PROGRAM VGR_State
VAR
	
	bStateIdle: BOOL := TRUE;
	bStatePlace: BOOL;
	bStateHoming: BOOL;
	bStatePick: BOOL;
	tolerance : UINT := 5;
	
	bInPositionPickVertical : BOOL;
	bInPositionPickHorizontal : BOOL;
	bInPositionPickRotate : BOOL;
	bInPositionPlaceVertical : BOOL;
	bInPositionPlaceHorizontal : BOOL;
	bInPositionPlaceRotate : BOOL;
	
	bValveClosed : BOOL;
	
	RS_Idle: RS;
	
	RS_Homing: RS;
	
	RS_Pick: RS;
	bValveOpened: BOOL;
	RS_Place: RS;
	bValveOpen: BOOL;
	SR_ESTOP: SR;
	bStateEStop: BOOL;
	AxisMovementController_Vertical: AxisMovementController;
	AxisMovementController_Horizontal: AxisMovementController;
	AxisReferencing_Vertical: AxisReferencing;
	AxisReferencing_Horizontal: AxisReferencing;
	AxisReferencing_Rotational: AxisReferencing;
	AxisMovementController_Rotation: AxisMovementController;
END_VAR
VAR // added by the converter: edge detectors and wires of the graphical bodies
    _w1 : BOOL;
END_VAR

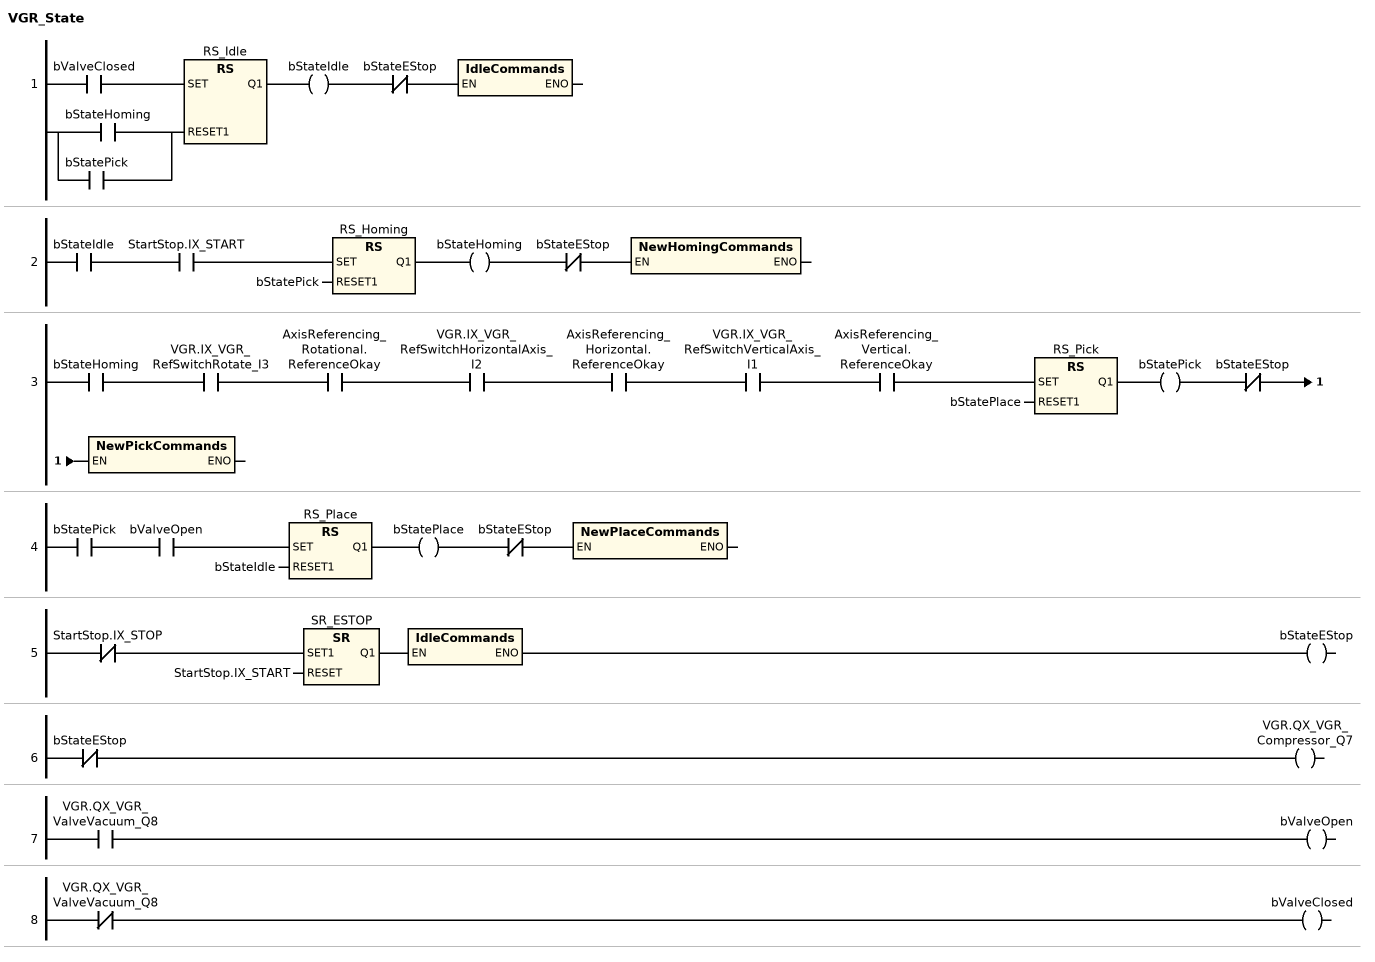
// NETWORK 1
RS_Idle(SET := bValveClosed, RESET1 := bStateHoming OR bStatePick); // RS
bStateIdle := RS_Idle.Q1;
IF RS_Idle.Q1 AND NOT bStateEStop THEN IdleCommands(); END_IF

// NETWORK 2
RS_Homing(SET := bStateIdle AND StartStop.IX_START, RESET1 := bStatePick); // RS
bStateHoming := RS_Homing.Q1;
IF RS_Homing.Q1 AND NOT bStateEStop THEN NewHomingCommands(); END_IF

// NETWORK 3
RS_Pick(SET := bStateHoming AND VGR.IX_VGR_RefSwitchRotate_I3 AND AxisReferencing_Rotational.ReferenceOkay AND VGR.IX_VGR_RefSwitchHorizontalAxis_I2 AND AxisReferencing_Horizontal.ReferenceOkay AND VGR.IX_VGR_RefSwitchVerticalAxis_I1 AND AxisReferencing_Vertical.ReferenceOkay, RESET1 := bStatePlace); // RS
bStatePick := RS_Pick.Q1;
IF RS_Pick.Q1 AND NOT bStateEStop THEN NewPickCommands(); END_IF

// NETWORK 4
RS_Place(SET := bStatePick AND bValveOpen, RESET1 := bStateIdle); // RS
bStatePlace := RS_Place.Q1;
IF RS_Place.Q1 AND NOT bStateEStop THEN NewPlaceCommands(); END_IF

// NETWORK 5
SR_ESTOP(SET1 := NOT StartStop.IX_STOP, RESET := StartStop.IX_START); // SR
_w1 := SR_ESTOP.Q1;
IF _w1 THEN IdleCommands(); END_IF
bStateEStop := _w1;

// NETWORK 6
VGR.QX_VGR_Compressor_Q7 := NOT bStateEStop;

// NETWORK 7
bValveOpen := VGR.QX_VGR_ValveVacuum_Q8;

// NETWORK 8
bValveClosed := NOT VGR.QX_VGR_ValveVacuum_Q8;

ACTION HomeCommands:
IF VGR.IX_VGR_RefSwitchVerticalAxis_I1 THEN
	VGR.QX_VGR_M1_VerticalAxisUp_Q1 := FALSE;
	VGR.QX_VGR_M1_VerticalAxisDown_Q2 := FALSE;
	VGR.QW_VGR_PWM_Vertical_Control := 0;
	VGR.QW_VGR_PWM_Vertical_M1 := 0;
	Encoder.setCounterVertical := TRUE;
	Encoder.setCounterValueVertical:= 0;
ELSE
	VGR.QX_VGR_M1_VerticalAxisUp_Q1 := TRUE;
	VGR.QX_VGR_M1_VerticalAxisDown_Q2 := FALSE;
	VGR.QW_VGR_PWM_Vertical_Control := 32;
	VGR.QW_VGR_PWM_Vertical_M1 := 5000;
END_IF
IF VGR.IX_VGR_RefSwitchHorizontalAxis_I2 THEN
	VGR.QX_VGR_M2_HorizontalAxisBackward_Q3 := FALSE;
    VGR.QX_VGR_M2_HorizontalAxisForward_Q4 := FALSE;
    VGR.QW_VGR_PWM_Horizontal_Control := 0;
    VGR.QW_VGR_PWM_Horizontal_M2 := 0;
	Encoder.setCounterHorizontal := TRUE;
ELSE
	VGR.QX_VGR_M2_HorizontalAxisBackward_Q3 := TRUE;
    VGR.QX_VGR_M2_HorizontalAxisForward_Q4 := FALSE;
    VGR.QW_VGR_PWM_Horizontal_Control := 32;
    VGR.QW_VGR_PWM_Horizontal_M2 := 5000;
END_IF
IF VGR.IX_VGR_RefSwitchHorizontalAxis_I2 THEN
	VGR.QX_VGR_M3_RotateClockwise_Q5 := FALSE;
    VGR.QX_VGR_M3_RotateCounterClockwise_Q6 := FALSE;
    VGR.QW_VGR_PWM_Rotate_Control := 0;
    VGR.QW_VGR_PWM_Rotate_M3 := 0;
	Encoder.setCounterRotate := TRUE;
ELSE
	VGR.QX_VGR_M3_RotateClockwise_Q5 := TRUE;
    VGR.QX_VGR_M3_RotateCounterClockwise_Q6 := FALSE;
    VGR.QW_VGR_PWM_Rotate_Control := 32;
    VGR.QW_VGR_PWM_Rotate_M3 := 5000;
END_IF
END_ACTION

ACTION IdleCommands:
VGR.QX_VGR_M1_VerticalAxisUp_Q1 := FALSE;
VGR.QX_VGR_M1_VerticalAxisDown_Q2 := FALSE;
VGR.QW_VGR_PWM_Vertical_Control := 0;
VGR.QW_VGR_PWM_Vertical_M1 := 0;
VGR.QX_VGR_M2_HorizontalAxisBackward_Q3 := FALSE;
VGR.QX_VGR_M2_HorizontalAxisForward_Q4 := FALSE;
VGR.QW_VGR_PWM_Horizontal_Control := 0;
VGR.QW_VGR_PWM_Horizontal_M2 := 0;
VGR.QX_VGR_M3_RotateClockwise_Q5 := FALSE;
VGR.QX_VGR_M3_RotateCounterClockwise_Q6 := FALSE;
VGR.QW_VGR_PWM_Rotate_Control := 0;
VGR.QW_VGR_PWM_Rotate_M3 := 0;
END_ACTION

ACTION NewHomingCommands:
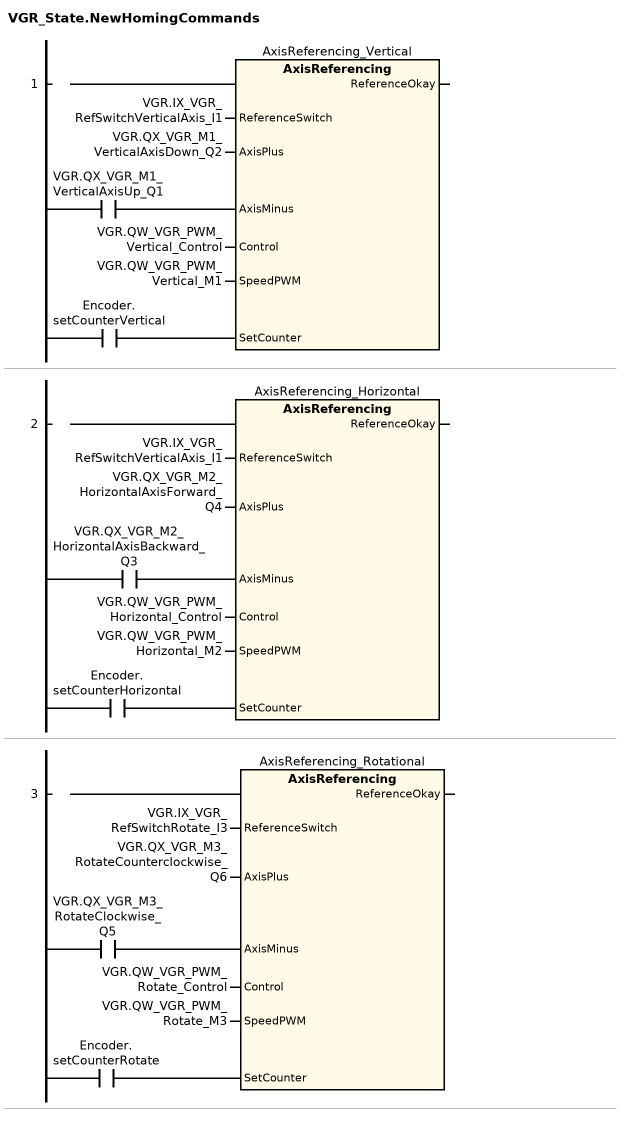
// NETWORK 1
AxisReferencing_Vertical(
    ReferenceSwitch := VGR.IX_VGR_RefSwitchVerticalAxis_I1,
    AxisPlus := VGR.QX_VGR_M1_VerticalAxisDown_Q2,
    AxisMinus := VGR.QX_VGR_M1_VerticalAxisUp_Q1,
    Control := VGR.QW_VGR_PWM_Vertical_Control,
    SpeedPWM := VGR.QW_VGR_PWM_Vertical_M1,
    SetCounter := Encoder.setCounterVertical); // AxisReferencing

// NETWORK 2
AxisReferencing_Horizontal(
    ReferenceSwitch := VGR.IX_VGR_RefSwitchVerticalAxis_I1,
    AxisPlus := VGR.QX_VGR_M2_HorizontalAxisForward_Q4,
    AxisMinus := VGR.QX_VGR_M2_HorizontalAxisBackward_Q3,
    Control := VGR.QW_VGR_PWM_Horizontal_Control,
    SpeedPWM := VGR.QW_VGR_PWM_Horizontal_M2,
    SetCounter := Encoder.setCounterHorizontal); // AxisReferencing

// NETWORK 3
AxisReferencing_Rotational(
    ReferenceSwitch := VGR.IX_VGR_RefSwitchRotate_I3,
    AxisPlus := VGR.QX_VGR_M3_RotateCounterclockwise_Q6,
    AxisMinus := VGR.QX_VGR_M3_RotateClockwise_Q5,
    Control := VGR.QW_VGR_PWM_Rotate_Control,
    SpeedPWM := VGR.QW_VGR_PWM_Rotate_M3,
    SetCounter := Encoder.setCounterRotate); // AxisReferencing
END_ACTION

ACTION NewPickCommands:
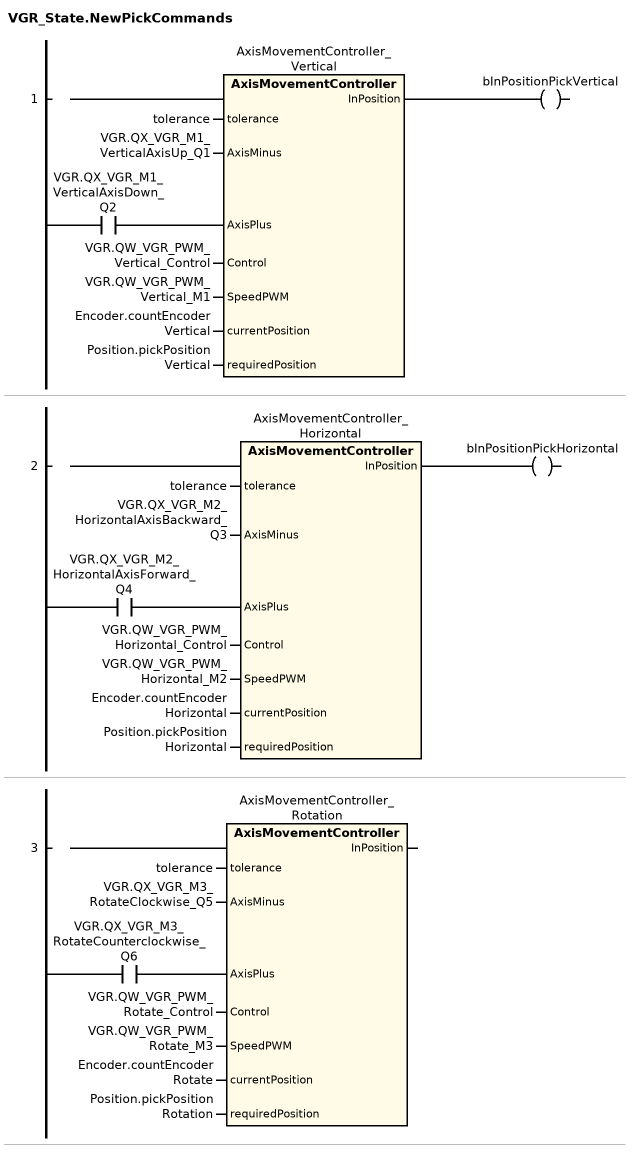
// NETWORK 1
AxisMovementController_Vertical(
    tolerance := tolerance,
    AxisMinus := VGR.QX_VGR_M1_VerticalAxisUp_Q1,
    AxisPlus := VGR.QX_VGR_M1_VerticalAxisDown_Q2,
    Control := VGR.QW_VGR_PWM_Vertical_Control,
    SpeedPWM := VGR.QW_VGR_PWM_Vertical_M1,
    currentPosition := Encoder.countEncoderVertical,
    requiredPosition := Position.pickPositionVertical); // AxisMovementController
bInPositionPickVertical := AxisMovementController_Vertical.InPosition;

// NETWORK 2
AxisMovementController_Horizontal(
    tolerance := tolerance,
    AxisMinus := VGR.QX_VGR_M2_HorizontalAxisBackward_Q3,
    AxisPlus := VGR.QX_VGR_M2_HorizontalAxisForward_Q4,
    Control := VGR.QW_VGR_PWM_Horizontal_Control,
    SpeedPWM := VGR.QW_VGR_PWM_Horizontal_M2,
    currentPosition := Encoder.countEncoderHorizontal,
    requiredPosition := Position.pickPositionHorizontal); // AxisMovementController
bInPositionPickHorizontal := AxisMovementController_Horizontal.InPosition;

// NETWORK 3
AxisMovementController_Rotation(
    tolerance := tolerance,
    AxisMinus := VGR.QX_VGR_M3_RotateClockwise_Q5,
    AxisPlus := VGR.QX_VGR_M3_RotateCounterclockwise_Q6,
    Control := VGR.QW_VGR_PWM_Rotate_Control,
    SpeedPWM := VGR.QW_VGR_PWM_Rotate_M3,
    currentPosition := Encoder.countEncoderRotate,
    requiredPosition := Position.pickPositionRotation); // AxisMovementController
END_ACTION

ACTION NewPlaceCommands:
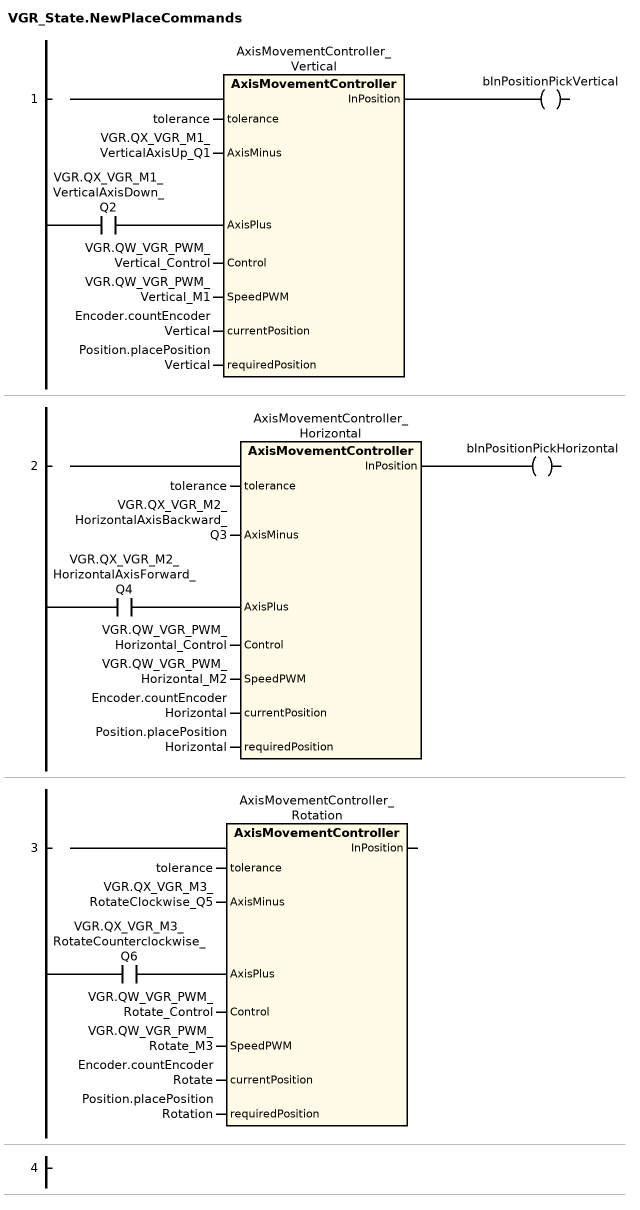
// NETWORK 1
AxisMovementController_Vertical(
    tolerance := tolerance,
    AxisMinus := VGR.QX_VGR_M1_VerticalAxisUp_Q1,
    AxisPlus := VGR.QX_VGR_M1_VerticalAxisDown_Q2,
    Control := VGR.QW_VGR_PWM_Vertical_Control,
    SpeedPWM := VGR.QW_VGR_PWM_Vertical_M1,
    currentPosition := Encoder.countEncoderVertical,
    requiredPosition := Position.placePositionVertical); // AxisMovementController
bInPositionPickVertical := AxisMovementController_Vertical.InPosition;

// NETWORK 2
AxisMovementController_Horizontal(
    tolerance := tolerance,
    AxisMinus := VGR.QX_VGR_M2_HorizontalAxisBackward_Q3,
    AxisPlus := VGR.QX_VGR_M2_HorizontalAxisForward_Q4,
    Control := VGR.QW_VGR_PWM_Horizontal_Control,
    SpeedPWM := VGR.QW_VGR_PWM_Horizontal_M2,
    currentPosition := Encoder.countEncoderHorizontal,
    requiredPosition := Position.placePositionHorizontal); // AxisMovementController
bInPositionPickHorizontal := AxisMovementController_Horizontal.InPosition;

// NETWORK 3
AxisMovementController_Rotation(
    tolerance := tolerance,
    AxisMinus := VGR.QX_VGR_M3_RotateClockwise_Q5,
    AxisPlus := VGR.QX_VGR_M3_RotateCounterclockwise_Q6,
    Control := VGR.QW_VGR_PWM_Rotate_Control,
    SpeedPWM := VGR.QW_VGR_PWM_Rotate_M3,
    currentPosition := Encoder.countEncoderRotate,
    requiredPosition := Position.placePositionRotation); // AxisMovementController

// NETWORK 4
END_ACTION

ACTION PickCommands:
IF  AboutEqual(IN1:= Encoder.countEncoderVertical,
	IN2:= Position.pickPositionVertical,
Tolerance:= tolerance)
 THEN
	VGR.QX_VGR_M1_VerticalAxisUp_Q1 := FALSE;
	VGR.QX_VGR_M1_VerticalAxisDown_Q2 := FALSE;
	VGR.QW_VGR_PWM_Vertical_Control := 0;
	VGR.QW_VGR_PWM_Vertical_M1 := 0;
	bInPositionPickVertical := TRUE;
ELSIF Encoder.countEncoderVertical > Position.pickPositionVertical AND NOT bInPositionPickVertical THEN
	VGR.QX_VGR_M1_VerticalAxisUp_Q1 := TRUE;
	VGR.QX_VGR_M1_VerticalAxisDown_Q2 := FALSE;
	VGR.QW_VGR_PWM_Vertical_Control := 32;
	VGR.QW_VGR_PWM_Vertical_M1 := 5000;
	bInPositionPickVertical := FALSE;
ELSE
	VGR.QX_VGR_M1_VerticalAxisUp_Q1 := FALSE;
	VGR.QX_VGR_M1_VerticalAxisDown_Q2 := TRUE;
	VGR.QW_VGR_PWM_Vertical_Control := 32;
	VGR.QW_VGR_PWM_Vertical_M1 := 5000;
	bInPositionPickVertical := FALSE;
END_IF
IF AboutEqual(IN1:= Encoder.countEncoderHorizontal,
	IN2:= Position.pickPositionHorizontal,
Tolerance:= tolerance) THEN
	VGR.QX_VGR_M2_HorizontalAxisBackward_Q3 := FALSE;
    VGR.QX_VGR_M2_HorizontalAxisForward_Q4 := FALSE;
    VGR.QW_VGR_PWM_Horizontal_Control := 0;
    VGR.QW_VGR_PWM_Horizontal_M2 := 0;
	bInPositionPickHorizontal := TRUE;
ELSIF Encoder.countEncoderHorizontal > Position.pickPositionHorizontal  AND NOT bInPositionPickHorizontal THEN
	VGR.QX_VGR_M2_HorizontalAxisBackward_Q3 := TRUE;
    VGR.QX_VGR_M2_HorizontalAxisForward_Q4 := FALSE;
    VGR.QW_VGR_PWM_Horizontal_Control := 32;
    VGR.QW_VGR_PWM_Horizontal_M2 := 5000;
	bInPositionPickHorizontal := FALSE;
ELSE
	VGR.QX_VGR_M2_HorizontalAxisBackward_Q3 := FALSE;
	VGR.QX_VGR_M2_HorizontalAxisForward_Q4 := TRUE;
	VGR.QW_VGR_PWM_Horizontal_Control := 32;
	VGR.QW_VGR_PWM_Horizontal_M2 := 5000;
	bInPositionPickHorizontal := FALSE;
END_IF
IF  AboutEqual(IN1:= Encoder.countEncoderRotate,
	IN2:= Position.pickPositionRotation,
Tolerance:= tolerance) THEN
    VGR.QX_VGR_M3_RotateClockwise_Q5 := FALSE;
    VGR.QX_VGR_M3_RotateCounterClockwise_Q6 := FALSE;
    VGR.QW_VGR_PWM_Rotate_Control := 0;
    VGR.QW_VGR_PWM_Rotate_M3 := 0;
	bInPositionPickRotate := TRUE;
ELSIF Encoder.countEncoderRotate > Position.pickPositionRotation  AND NOT bInPositionPickRotate THEN
	VGR.QX_VGR_M3_RotateClockwise_Q5 := FALSE;
    VGR.QX_VGR_M3_RotateCounterClockwise_Q6 := TRUE;
    VGR.QW_VGR_PWM_Rotate_Control := 32;
    VGR.QW_VGR_PWM_Rotate_M3 := 5000;
	bInPositionPickRotate := FALSE;
ELSE
	VGR.QX_VGR_M3_RotateClockwise_Q5 := TRUE;
    VGR.QX_VGR_M3_RotateCounterClockwise_Q6 := FALSE;
    VGR.QW_VGR_PWM_Rotate_Control := 32;
    VGR.QW_VGR_PWM_Rotate_M3 := 5000;
	bInPositionPickRotate := FALSE;
END_IF

IF bInPositionPickRotate AND bInPositionPickRotate AND bInPositionPickRotate THEN
	VGR.QX_VGR_ValveVacuum_Q8 := TRUE;
ELSE
	VGR.QX_VGR_ValveVacuum_Q8 := FALSE;
END_IF
END_ACTION

ACTION PlaceCommands:
IF  Encoder.countEncoderVertical = Position.placePositionVertical OR
	(Position.pickPositionVertical+tolerance > Encoder.countEncoderVertical OR 
	Encoder.countEncoderVertical > Position.pickPositionVertical-tolerance ) THEN
	VGR.QX_VGR_M1_VerticalAxisUp_Q1 := FALSE;
	VGR.QX_VGR_M1_VerticalAxisDown_Q2 := FALSE;
	VGR.QW_VGR_PWM_Vertical_Control := 0;
	VGR.QW_VGR_PWM_Vertical_M1 := 0;
	bInPositionPlaceVertical := TRUE;
ELSIF Encoder.countEncoderVertical > Position.placePositionVertical THEN
	VGR.QX_VGR_M1_VerticalAxisUp_Q1 := FALSE;
	VGR.QX_VGR_M1_VerticalAxisDown_Q2 := TRUE;
	VGR.QW_VGR_PWM_Vertical_Control := 32;
	VGR.QW_VGR_PWM_Vertical_M1 := 5000;
	bInPositionPlaceVertical := FALSE;
ELSE
	VGR.QX_VGR_M1_VerticalAxisUp_Q1 := TRUE;
	VGR.QX_VGR_M1_VerticalAxisDown_Q2 := FALSE;
	VGR.QW_VGR_PWM_Vertical_Control := 32;
	VGR.QW_VGR_PWM_Vertical_M1 := 5000;
	bInPositionPlaceVertical := FALSE;
END_IF
IF Encoder.countEncoderHorizontal = Position.placePositionHorizontal OR 
(Encoder.countEncoderHorizontal < Position.pickPositionHorizontal + tolerance)OR 
(Encoder.countEncoderHorizontal > Position.pickPositionHorizontal -tolerance) THEN
	VGR.QX_VGR_M2_HorizontalAxisBackward_Q3 := FALSE;
    VGR.QX_VGR_M2_HorizontalAxisForward_Q4 := FALSE;
    VGR.QW_VGR_PWM_Horizontal_Control := 0;
    VGR.QW_VGR_PWM_Horizontal_M2 := 0;
	bInPositionPlaceHorizontal := TRUE;
ELSIF Encoder.countEncoderHorizontal > Position.placePositionHorizontal THEN
	VGR.QX_VGR_M2_HorizontalAxisBackward_Q3 := TRUE;
    VGR.QX_VGR_M2_HorizontalAxisForward_Q4 := FALSE;
    VGR.QW_VGR_PWM_Horizontal_Control := 32;
    VGR.QW_VGR_PWM_Horizontal_M2 := 5000;
	bInPositionPlaceHorizontal := FALSE;
ELSE
	VGR.QX_VGR_M2_HorizontalAxisBackward_Q3 := FALSE;
	VGR.QX_VGR_M2_HorizontalAxisForward_Q4 := TRUE;
	VGR.QW_VGR_PWM_Horizontal_Control := 32;
	VGR.QW_VGR_PWM_Horizontal_M2 := 5000;
	bInPositionPlaceHorizontal := FALSE;
END_IF
IF  Encoder.countEncoderRotate=Position.placePositionRotation  OR 
(Encoder.countEncoderRotate < Position.pickPositionRotation+tolerance) OR 
(Encoder.countEncoderRotate>Position.pickPositionRotation-tolerance) THEN
    VGR.QX_VGR_M3_RotateClockwise_Q5 := FALSE;
    VGR.QX_VGR_M3_RotateCounterClockwise_Q6 := FALSE;
    VGR.QW_VGR_PWM_Rotate_Control := 0;
    VGR.QW_VGR_PWM_Rotate_M3 := 0;
	bInPositionPlaceRotate := TRUE;
ELSIF Encoder.countEncoderRotate > Position.placePositionRotation THEN
	VGR.QX_VGR_M3_RotateClockwise_Q5 := FALSE;
    VGR.QX_VGR_M3_RotateCounterClockwise_Q6 := TRUE;
    VGR.QW_VGR_PWM_Rotate_Control := 32;
    VGR.QW_VGR_PWM_Rotate_M3 := 5000;
	bInPositionPlaceRotate := FALSE;
ELSE
	VGR.QX_VGR_M3_RotateClockwise_Q5 := TRUE;
    VGR.QX_VGR_M3_RotateCounterClockwise_Q6 := FALSE;
    VGR.QW_VGR_PWM_Rotate_Control := 32;
    VGR.QW_VGR_PWM_Rotate_M3 := 5000;
	bInPositionPlaceRotate := FALSE;
END_IF

IF bInPositionPlaceHorizontal AND bInPositionPlaceRotate AND bInPositionPlaceVertical THEN
	VGR.QX_VGR_ValveVacuum_Q8 := FALSE;
ELSE
	VGR.QX_VGR_ValveVacuum_Q8 := TRUE;
END_IF
END_ACTION

END_PROGRAM

(* stored: Version 1.1.0.1, ProductVersion 3.1.4024.12
   POU VGR_State: Id {7aa8a406-b458-426c-9530-cc62a1b42f8a}, SpecialFunc None
   Action HomeCommands: Id {0f636ef8-07f3-4884-a7a6-370109e8cfaa}
   Action IdleCommands: Id {c22b6015-031e-44d1-9a49-ef0c9e3c7f44}
   Action NewHomingCommands: Id {56950258-6488-4c40-9d15-434b1ca9d02a}
   Action NewPickCommands: Id {c336029e-b54d-4c80-b2f9-8cac11d6896b}
   Action NewPlaceCommands: Id {43b75217-0a31-4d31-9610-cf6accadfee8}
   Action PickCommands: Id {dc673986-ad1f-4d3b-a207-aacd8963d3f2}
   Action PlaceCommands: Id {975bda5b-711b-4685-8fbc-c7b3b107ef25} *)
